Fanuc KAREL source: kt00443.KL

-- PROVISIONAL review KL for V940-1; original PC SHA256 7884fb90572bccd125b3ab85da2b6448fed229100b2cc2202ee92744ff1276d0
-- Incomplete behavior may be omitted. Consult companion uncertainty JSON. Do not deploy.
PROGRAM KT00443
%NOLOCKGROUP
VAR
  R1 : REAL
  OUT : BOOLEAN
-- UNRESOLVED_DECL Y2 type=002018
BEGIN
  -- V9_ZERO_TABLE_METADATA_HINT layout=0001; no indexed target words; source/name/runtime held
  -- UNRESOLVED_PC offsets 5-16; opcodes 2E,23
  -- UNRESOLVED_PC offsets 21-35; opcodes 2E,22,9D,33,B2
  -- UNRESOLVED_PC offsets 40-63; opcodes 21,22,9D,33,B1,64,72,23
  -- UNRESOLVED_PC offsets 68-72; opcodes 7F
END KT00443
